Xinje XDPPro project, PLC1: XD3-16 (software 3.7.17b 2023-10-13)

PROGRAM Ladder

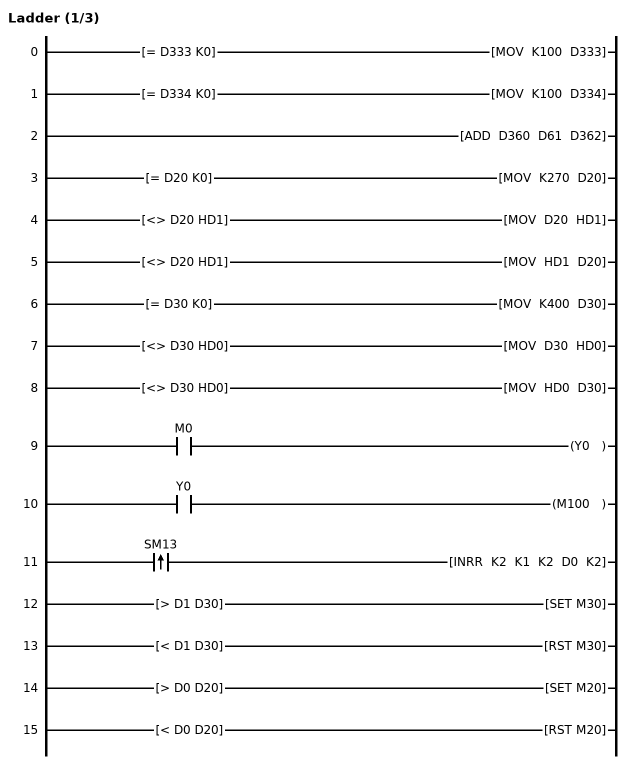
LD=    D333 K0
MOV    K100 D333
LD=    D334 K0
MOV    K100 D334
ADD    D360 D61 D362
LD=    D20 K0
MOV    K270 D20
LD<>   D20 HD1
MOV    D20 HD1
LD<>   D20 HD1
MOV    HD1 D20
LD=    D30 K0
MOV    K400 D30
LD<>   D30 HD0
MOV    D30 HD0
LD<>   D30 HD0
MOV    HD0 D30
LD     M0
OUT    Y0
LD     Y0
OUT    M100
LDP    SM13
INRR   K2 K1 K2 D0 K2
LD>    D1 D30
SET    M30
LD<    D1 D30
RST    M30
LD>    D0 D20
SET    M20
LD<    D0 D20
RST    M20

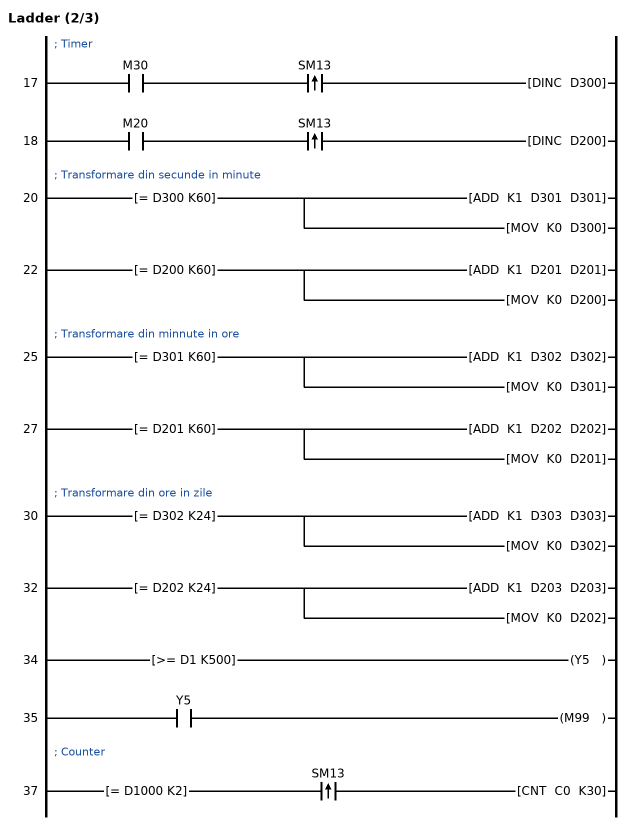
; Timer
LD     M30
ANDP   SM13
DINC   D300
LD     M20
ANDP   SM13
DINC   D200
; Transformare din secunde in minute
LD=    D300 K60
ADD    K1 D301 D301
MOV    K0 D300
LD=    D200 K60
ADD    K1 D201 D201
MOV    K0 D200
; Transformare din minnute in ore
LD=    D301 K60
ADD    K1 D302 D302
MOV    K0 D301
LD=    D201 K60
ADD    K1 D202 D202
MOV    K0 D201
; Transformare din ore in zile
LD=    D302 K24
ADD    K1 D303 D303
MOV    K0 D302
LD=    D202 K24
ADD    K1 D203 D203
MOV    K0 D202
LD>=   D1 K500
OUT    Y5
LD     Y5
OUT    M99
; Counter
LD=    D1000 K2
ANDP   SM13
CNT    C0 K30

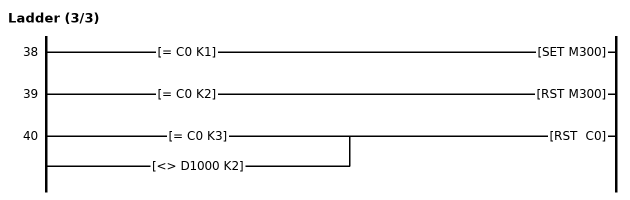
LD=    C0 K1
SET    M300
LD=    C0 K2
RST    M300
LD=    C0 K3
OR<>   D1000 K2
RST    C0